METHOD PRIVATE CreatePrototype : I_NodePrototype
VAR_INPUT
	PrototypePath : T_MAXSTRING;
	PrototypeNode : I_Node;
END_VAR
VAR
	pNodePrototype : POINTER TO NodePrototype;
END_VAR
pNodePrototype := __NEW(NodePrototype(Path := PrototypePath, Node := PrototypeNode));
CreatePrototype := pNodePrototype^;
END_METHOD

METHOD PRIVATE DisposeSelfCreatedNodePrototypes : BOOL
VAR
	prototype : I_NodePrototype;
END_VAR
WHILE selfCreatedPrototypes.TryPop(prototype) DO
	prototype.Dispose();
END_WHILE
END_METHOD

METHOD PUBLIC Accept
VAR_INPUT
	visitor : I_NodePrototypeVisitor;
END_VAR
VAR
	enumerator : I_ForwardEnumerator;
	nodePrototype : I_NodePrototype;
END_VAR
enumerator := prototypes.GetEnumerator();

WHILE enumerator.MoveNext() DO
	
	IF enumerator.TryGet(nodePrototype) THEN
		nodePrototype.Accept(Visitor);
	END_IF

END_WHILE

enumerator.Dispose();
END_METHOD

METHOD AddNodeAsPrototype : I_NodePrototype
VAR_INPUT
	Path : T_MAXSTRING;
	Node : I_Node;
END_VAR
VAR
	prototype : I_NodePrototype;
END_VAR
prototype := CreatePrototype(Path, Node);
selfCreatedPrototypes.Push(prototype);
AddNodePrototype(prototype);
AddNodeAsPrototype := prototype;
END_METHOD

METHOD PUBLIC AddNodePrototype
VAR_INPUT
	NodePrototype : I_NodePrototype;
END_VAR
prototypes.AddOrUpdate(NodePrototype.Path, NodePrototype);
END_METHOD

PROPERTY PUBLIC HasNodePrototypes : BOOL
GET
HasNodePrototypes := prototypes.Count > 0;
END_GET
END_PROPERTY

METHOD PUBLIC TryGetNodePrototypeByPath : BOOL
VAR_INPUT
	Path : T_MAXSTRING;
	Destination : REFERENCE TO I_NodePrototype;
END_VAR
VAR
	nodePrototype : I_NodePrototype;
END_VAR
IF NOT prototypes.TryGetValue(Path, nodePrototype) THEN
	RETURN;
END_IF

Destination := nodePrototype;
TryGetNodePrototypeByPath := TRUE;
END_METHOD

END_FUNCTION_BLOCK

// Node/Host/NodeHost
{attribute 'linkalways'} 
{attribute 'no_explicit_call' := 'This FB is a CLASS and must be accessed using methods or properties'}
{attribute 'enable_dynamic_creation'}
FUNCTION_BLOCK NodeHost IMPLEMENTS I_Nodes, I_Serializable
VAR
	hostParent : I_HostNodes;
	eventTarget : I_EventTarget;
	nodes : Dictionary;
	nodesInOrder : LinkedList;
END_VAR

METHOD FB_init : BOOL
VAR_INPUT
	bInitRetains : BOOL; // if TRUE, the retain variables are initialized (warm start / cold start)
	bInCopyCode : BOOL;  // if TRUE, the instance afterwards gets moved into the copy code (online change)
	Parent : I_HostNodes;
	parentEventTarget : I_EventTarget;
END_VAR
hostParent := Parent;
eventTarget := parentEventTarget;
END_METHOD

METHOD PROTECTED EmitOnNodeAddedEvent
VAR_INPUT
	Node : I_Node;
END_VAR
VAR
	pNodeAddedEvent : POINTER TO NodeAddedEvent;
END_VAR
IF eventTarget = 0 THEN
	RETURN;
END_IF

pNodeAddedEvent := __NEW(NodeAddedEvent(Target := Node));
eventTarget.Emit('OnNodeAdded',pNodeAddedEvent^);
pNodeAddedEvent^.Dispose();
END_METHOD

METHOD PROTECTED UpdateExecutionOrder
VAR_INPUT
	Node : I_Node;
END_VAR
VAR
	currentPosition : I_LinkedListNode;
	currentNode : I_Node;
END_VAR
// is the list empty?
IF nodesInOrder.First = 0 THEN
	// if so, add our node first and jump out as done.
	nodesInOrder.AddFirst(Node);
	RETURN;
END_IF

// if not empty, then is our node higher priorty than the first in the list. 
NodesInOrder.First.TryGet(currentNode); 
IF currentNode.Order > Node.Order THEN
	// if yes, we are now first, jump out as done. 
	nodesInOrder.AddFirst(Node);
	RETURN;
END_IF

// here, the list has something in it, and we have less priority than the node in first place.

// get the last node in the list and remember this as "currentPosition" 
currentPosition := nodesInOrder.Last;

WHILE (TRUE) DO
	
	currentPosition.TryGet(currentNode); 
	// is the current position higer priority than our node?
	IF currentNode.Order <= Node.Order THEN
		// if so, then we go after, jump out as we are done. 
		nodesInOrder.AddAfter(currentPosition, Node);
		RETURN;
	END_IF
	
	// move one up the list towards the top and try again.
	currentPosition := currentPosition.Previous;

END_WHILE
END_METHOD

METHOD PUBLIC Accept
VAR_INPUT
	Visitor : I_NodeVisitor;
END_VAR
VAR
	enumerator : I_ForwardEnumerator;
	node : I_Node;
END_VAR
enumerator := nodes.GetEnumerator();

WHILE (enumerator.MoveNext()) DO
	
	IF enumerator.TryGet(node) THEN
		node.Accept(Visitor);
	END_IF

END_WHILE

enumerator.Dispose();
END_METHOD

METHOD PUBLIC AddNode
VAR_INPUT
	Node : I_Node;
END_VAR
nodes.AddOrUpdate(Node.id, Node);
UpdateExecutionOrder(Node);
EmitOnNodeAddedEvent(Node);
END_METHOD

METHOD PUBLIC Execute
VAR_INPUT
END_VAR
VAR
	enumerator : I_ForwardEnumerator;
	node : I_Node;
END_VAR
enumerator := nodesInOrder.GetEnumerator();

WHILE enumerator.MoveNext() DO
	IF enumerator.TryGet(node) THEN
		node.Execute();
	END_IF
END_WHILE

enumerator.Dispose();
END_METHOD

PROPERTY PUBLIC HasNodes : BOOL
GET
HasNodes := nodes.Count > 0;
END_GET
END_PROPERTY

METHOD PUBLIC RemoveNode
VAR_INPUT
	Node : I_Node;
END_VAR
nodes.Remove(Node.Id);
nodesInOrder.Remove(Node);
END_METHOD

METHOD PUBLIC SerializeWith
VAR_INPUT
	Serializer : I_Serializer;
END_VAR
VAR
	enumerator : I_ForwardEnumerator;
	node : I_Node;
END_VAR
IF nodes.Count = 0 THEN
	RETURN;
END_IF

Serializer.AddKey('nodes');
Serializer.StartArray();

enumerator := nodes.GetEnumerator();

WHILE enumerator.MoveNext() DO
	IF enumerator.TryGet(node) THEN
		node.SerializeWith(Serializer);
	END_IF
END_WHILE

Serializer.EndArray();
enumerator.Dispose();
END_METHOD

METHOD PUBLIC TryDeserializeFrom : BOOL
VAR_INPUT
	Deserializer : I_Deserializer;
	Feedback : I_DeserializerFeedback;
END_VAR
VAR
	nodeDeserializer : I_Deserializer;
	nodesEnumerator : I_DeserializerArrayForwardEnumerator;
	nodeId : T_MAXSTRING;
	node : I_Node;
END_VAR
nodeDeserializer := Deserializer.GetKeyArray('nodes');
nodesEnumerator := nodeDeserializer.GetArrayEnumerator();

WHILE nodesEnumerator.MoveNext() DO
	
	IF NOT nodesEnumerator.Current.TryGetKeyString('id',nodeId, Feedback) THEN
		CONTINUE;
	END_IF
	
	IF NOT TryGetNodeById(nodeId, node)THEN
		CONTINUE;
	END_IF
	
	node.TryDeserializeFrom(nodesEnumerator.Current, Feedback);

END_WHILE

nodesEnumerator.Dispose();
END_METHOD

METHOD PUBLIC TryGetNodeById : BOOL
VAR_INPUT
	Id : T_MAXSTRING;
	Destination : REFERENCE TO I_Node;
END_VAR
VAR
	node : I_Node;
END_VAR
IF NOT nodes.TryGetValue(Id, node) THEN
	RETURN;
END_IF

Destination := node;
TryGetNodeById := TRUE;
END_METHOD

END_FUNCTION_BLOCK

// Node/Events/NodeAddedEvent
{attribute 'linkalways'} 
{attribute 'no_explicit_call' := 'This FB is a CLASS and must be accessed using methods or properties'}
{attribute 'enable_dynamic_creation'}
FUNCTION_BLOCK NodeAddedEvent EXTENDS Disposable IMPLEMENTS I_NodeAddedEvent
VAR
	_target : I_Node;
END_VAR

METHOD FB_init : BOOL
VAR_INPUT
	bInitRetains : BOOL; // if TRUE, the retain variables are initialized (warm start / cold start)
	bInCopyCode : BOOL;  // if TRUE, the instance afterwards gets moved into the copy code (online change)
	Target : I_Node;
END_VAR
This^._target := Target;
END_METHOD

PROPERTY PUBLIC Target : I_Node
GET
Target := _target;
END_GET
END_PROPERTY

END_FUNCTION_BLOCK

// Node/Events/I_NodeAddedEvent
INTERFACE I_NodeAddedEvent EXTENDS I_Event

PROPERTY PUBLIC Target : I_Node
GET
END_GET
END_PROPERTY

END_INTERFACE

// Graph/Events/GraphAddedEvent
{attribute 'linkalways'} 
{attribute 'no_explicit_call' := 'This FB is a CLASS and must be accessed using methods or properties'}
{attribute 'enable_dynamic_creation'}
FUNCTION_BLOCK GraphAddedEvent EXTENDS Disposable IMPLEMENTS I_GraphAddedEvent
VAR
	_target : I_Graph;
END_VAR

METHOD FB_init : BOOL
VAR_INPUT
	bInitRetains : BOOL; // if TRUE, the retain variables are initialized (warm start / cold start)
	bInCopyCode : BOOL;  // if TRUE, the instance afterwards gets moved into the copy code (online change)
	Target : I_Graph;
END_VAR
This^._target := Target;
END_METHOD

PROPERTY PUBLIC Target : I_Graph
GET
Target := _target;
END_GET
END_PROPERTY

END_FUNCTION_BLOCK

// Graph/Events/I_GraphAddedEvent
INTERFACE I_GraphAddedEvent EXTENDS I_Event

PROPERTY PUBLIC Target : I_Graph
GET
END_GET
END_PROPERTY

END_INTERFACE

// Graph/Host/GraphHost
{attribute 'linkalways'} 
{attribute 'no_explicit_call' := 'This FB is a CLASS and must be accessed using methods or properties'}
{attribute 'enable_dynamic_creation'}
FUNCTION_BLOCK GraphHost IMPLEMENTS I_Graphs, I_Serializable
VAR
	hostParent : I_HostGraphs;
	eventTarget : I_EventTarget;
	graphs : Dictionary;	
END_VAR

METHOD FB_init : BOOL
VAR_INPUT
	bInitRetains : BOOL; // if TRUE, the retain variables are initialized (warm start / cold start)
	bInCopyCode : BOOL;  // if TRUE, the instance afterwards gets moved into the copy code (online change)
	Parent : I_HostGraphs;
	ParentEventTarget : I_EventTarget;
END_VAR
hostParent := Parent;
eventTarget := parentEventTarget;
END_METHOD

METHOD PROTECTED EmitOnGraphAddedEvent
VAR_INPUT
	Graph : I_Graph;
END_VAR
VAR
	pGraphAddedEvent : POINTER TO GraphAddedEvent;
END_VAR
IF eventTarget = 0 THEN
	RETURN;
END_IF

pGraphAddedEvent := __NEW(GraphAddedEvent(Target := Graph));
eventTarget.Emit('OnGraphAdded',pGraphAddedEvent^);
pGraphAddedEvent^.Dispose();
END_METHOD

METHOD PUBLIC Accept
VAR_INPUT
	visitor : I_GraphVisitor;
END_VAR
VAR
	enumerator : I_ForwardEnumerator;
	graph : I_Graph;
END_VAR
enumerator := graphs.GetEnumerator();

WHILE (enumerator.MoveNext()) DO
	
	IF enumerator.TryGet(graph) THEN
		graph.Accept(Visitor);
	END_IF

END_WHILE

enumerator.Dispose();
END_METHOD

METHOD PUBLIC AddGraph
VAR_INPUT
	Graph : I_Graph;
END_VAR
graphs.AddOrUpdate(Graph.Uuid, Graph);
EmitOnGraphAddedEvent(Graph);
END_METHOD

METHOD PUBLIC DisposeAll
VAR_INPUT
END_VAR
VAR
	enumerator : I_ForwardEnumerator;
	graph : I_Graph;
END_VAR
enumerator := graphs.GetEnumerator();

WHILE enumerator.MoveNext() DO
	IF enumerator.TryGet(graph) THEN
		graph.Dispose();
	END_IF
END_WHILE

graphs.Clear();

enumerator.Dispose();
END_METHOD

METHOD PUBLIC Execute
VAR_INPUT
END_VAR
VAR
	enumerator : I_ForwardEnumerator;
	graph : I_Graph;
END_VAR
enumerator := graphs.GetEnumerator();

WHILE enumerator.MoveNext() DO
	IF enumerator.TryGet(graph) THEN
		graph.Execute();
	END_IF
END_WHILE

enumerator.Dispose();
END_METHOD

METHOD PUBLIC RemoveGraph
VAR_INPUT
	Graph : I_Graph;
END_VAR
graphs.Remove(Graph.Uuid);
END_METHOD

METHOD PUBLIC SerializeWith
VAR_INPUT
	Serializer : I_Serializer;
END_VAR
VAR
	enumerator : I_ForwardEnumerator;
	graph : I_Graph;
END_VAR
IF graphs.Count = 0 THEN
	RETURN;
END_IF

Serializer.AddKey('graphs');
Serializer.StartArray();

enumerator := graphs.GetEnumerator();

WHILE enumerator.MoveNext() DO
	IF enumerator.TryGet(graph) THEN
		graph.SerializeWith(Serializer);
	END_IF
END_WHILE

Serializer.EndArray();
enumerator.Dispose();
END_METHOD

METHOD PUBLIC TryGetGraphByUuid : BOOL
VAR_INPUT
	Uuid : T_MAXSTRING;
	Destination : REFERENCE TO I_Graph;
END_VAR
VAR
	graph : I_Graph;
END_VAR
IF NOT graphs.TryGetValue(Uuid, graph) THEN
	RETURN;
END_IF

Destination := graph;
TryGetGraphByUuid := TRUE;
END_METHOD

END_FUNCTION_BLOCK

// Graph/Interfaces/I_Graphs
INTERFACE I_Graphs

METHOD PUBLIC Accept
VAR_INPUT
	visitor : I_GraphVisitor;
END_VAR
END_METHOD

METHOD PUBLIC AddGraph
VAR_INPUT
	Graph : I_Graph;
END_VAR
END_METHOD

METHOD PUBLIC DisposeAll
VAR_INPUT
END_VAR
END_METHOD

METHOD PUBLIC Execute
VAR_INPUT
END_VAR
END_METHOD

METHOD PUBLIC RemoveGraph
VAR_INPUT
	Graph : I_Graph;
END_VAR
END_METHOD

METHOD PUBLIC TryGetGraphByUuid : BOOL
VAR_INPUT
	Uuid : T_MAXSTRING;
	Destination : REFERENCE TO I_Graph;
END_VAR
END_METHOD

END_INTERFACE

// Graph/Interfaces/I_HostGraphs
INTERFACE I_HostGraphs

PROPERTY Graphs : I_Graphs
GET
END_GET
END_PROPERTY

END_INTERFACE

// GraphFramework/Interface/I_GraphFramework
INTERFACE I_GraphFramework

METHOD PUBLIC Create : I_Graph
VAR_INPUT
END_VAR
END_METHOD

PROPERTY PUBLIC Datatypes : I_Datatypes
GET
END_GET
END_PROPERTY

PROPERTY PUBLIC NodeFactory : I_NodeFactory
GET
END_GET
END_PROPERTY

END_INTERFACE

// GraphFramework/GraphFramework
{attribute 'linkalways'} 
{attribute 'no_explicit_call' := 'This FB is a CLASS and must be accessed using methods or properties'}
{attribute 'enable_dynamic_creation'}
FUNCTION_BLOCK GraphFramework IMPLEMENTS I_GraphFramework
VAR
	_nodeFactory : NodeFactory;
	_datatypes : Datatypes;
END_VAR

METHOD PUBLIC Create : I_Graph
VAR
	pGraph : POINTER TO Graph;
END_VAR
pGraph := __NEW(Graph(NodeFactory := _nodeFactory));
Create := pGraph^;
END_METHOD

PROPERTY PUBLIC Datatypes : I_Datatypes
GET
Datatypes := _datatypes;
END_GET
END_PROPERTY

METHOD PUBLIC InstallDatatypePack
VAR_INPUT
	DatatypePack : I_DatatypePack;
END_VAR
DatatypePack.RegisterWith(Datatypes);
END_METHOD

METHOD PUBLIC InstallNodePack
VAR_INPUT
	NodePack : I_NodePack;
END_VAR
NodePack.RegisterWithNodeFactory(NodeFactory);
END_METHOD

PROPERTY PUBLIC NodeFactory : I_NodeFactory
GET
NodeFactory := _nodeFactory;
END_GET
END_PROPERTY

END_FUNCTION_BLOCK

// NodePack/I_NodePack
INTERFACE I_NodePack

METHOD PUBLIC RegisterWithNodeFactory
VAR_INPUT
	NodeFactory : I_NodeFactory;
END_VAR
END_METHOD

END_INTERFACE
